// TIA Portal V20 export
VAR_GLOBAL   // PLC tag table "CentralFunctions"
END_VAR
VAR_GLOBAL CONSTANT   // user constants
   MAX_NO_OF_DEVICES_X1 : Int := 100;
   MAX_NO_OF_MODULES_X1 : Int := 100;
   MAX_NO_OF_DEVICES_X2 : Int := 100;
   MAX_NO_OF_MODULES_X2 : Int := 100;
END_VAR
